PROGRAM P3_04_Alarms
VAR 
	fbEventLogger		:FB_TcEventLogger;
	fbCsvExportSetting	:FB_TcEventCsvExportSettings;
	fbExportFilter		:FB_TcEventFilter;

	fbTrig				:R_TRIG;
	
	ulFilter1			:ULINT;
	ulFilter2			:ULINT;
	
	sPath				:STRING;
	
	
END_VAR

//Link here...

ulFilter1:=P3_01_BatchData.ulBatchOpen;
ulFilter2:=P3_01_BatchData.ulBatchClose;

fbTrig(CLK:=GV.stReport.bExport_Alarms);
IF GV.stReport.bExport_Alarms THEN
	IF fbTrig.Q THEN
		fbCsvExportSetting.Clear();
		fbCsvExportSetting.bWithHeader:=TRUE;
		fbCsvExportSetting.sDelimiter:=',';
		fbCsvExportSetting.AddFilter(fbExportFilter);
		fbExportFilter.Clear();
		fbExportFilter.IsAlarm().AND_OP().
		TimeRaised.GreaterThanOrEqualTo(ulFilter1).AND_OP().
		TimeRaised.LessThanOrEqualTo(ulFilter2).AND_OP().
		Source.Name.EqualTo('GV.stAlarm');
	END_IF
	
	sPath:=CONCAT(CONST.PROJECT_DIR,'Reports\1. Raw Data\AlarmLog.txt');
	
	IF fbEventLogger.ExportLoggedEvents(sPath,fbCsvExportSetting) THEN
		GV.stReport.bExport_Alarms:=FALSE;
	END_IF
END_IF

END_PROGRAM

(* stored: Version 1.1.0.1, ProductVersion 3.1.4024.12
   POU P3_04_Alarms: Id {6413df8d-b0e8-453f-b184-6acee373b8ea}, SpecialFunc None *)
